TYPE ST_SYSTEM_MachineMode :
STRUCT
	bDisable			: BOOL;
	bManual			: BOOL;
	bAutomatic		:  BOOL;
END_STRUCT
END_TYPE

(* stored: Version 1.1.0.1, ProductVersion 3.1.4024.15
   DUT ST_SYSTEM_MachineMode: Id {2f45629e-eceb-4fd7-981e-dd744aa28a3e} *)
